ABB RobotStudio station: material handling 06 03 2024 guna basith_1.rsstn

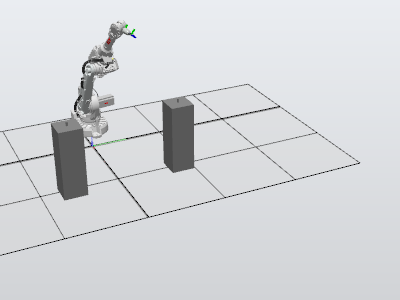
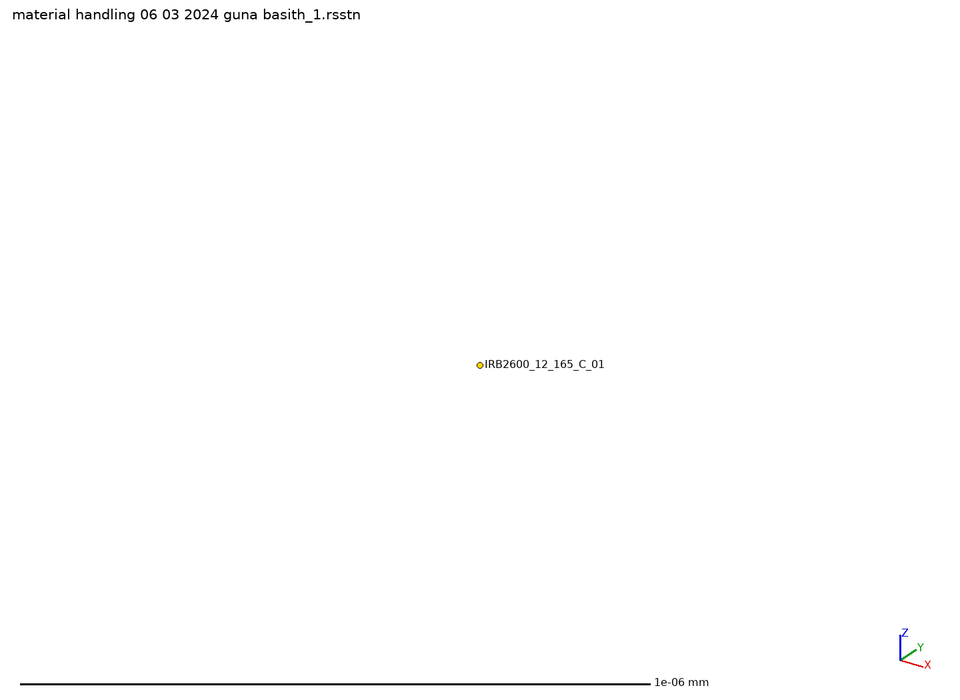
[picture v1: parts stored in the station drawn from their meshes, with robot base, taught points and paths (robot models come from the ABB library and are not in the file)]
Station Station (saved by RobotStudio 23.4.10609.1)
Controller Controller16, task T_ROB1: task frame (RAPID world) sits at (0, 0, 245) mm in the station
Controller Controller16
  mechanical unit ROB_1: IRB2600_12_165_C_01, 6 joints, base frame (0, 0, 0) mm
Layout (positions relative to the parent item):
  - Concrete [part, from Dispencing\Concrete.rslib]
  - IRB2600_12_165_C_01 [mechanism, from %ABB.RobotStudio.Models.IRB2600%\IRB2600_12_165_C_01.rslib] at (0, 0, 245) mm; joint values [0.1438, 0.4918, -1.2873, 3.4677, -1.1118, 3.9518] (rad or m)
  - SmartComponent_3 [smart component] at (1018.61, 172.16, 1931.71) mm, rotated rx 108.49 ry 28.78 rz 124.78 deg
      signals: DI attach
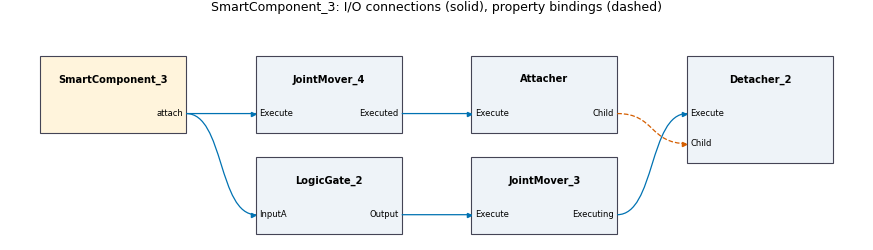
      connections:
        SmartComponent_3.attach -> JointMover_4.Execute
        JointMover_4.Executed -> Attacher.Execute
        SmartComponent_3.attach -> LogicGate_2.InputA
        LogicGate_2.Output -> JointMover_3.Execute
        JointMover_3.Executing -> Detacher_2.Execute
        Attacher.Child => Detacher_2.Child
    - Smart_Gripper_Servo_Fingers [mechanism, from %ABB.RobotStudio.Models.SmartGripper%\ABB_Smart_Gripper_Servo_Fingers.rslib] at (0, 0, 0) mm; joint values [0.023] (rad or m)
    - JointMover_3 [smart component, from Components\JointMover.rslib]
        properties: Mechanism=Smart_Gripper_Servo_Fingers; Relative=false; Duration=0; J1=0.024
    - JointMover_4 [smart component, from Components\JointMover.rslib]
        properties: Mechanism=Smart_Gripper_Servo_Fingers; Relative=false; Duration=0; J1=0.023
    - Detacher_2 [smart component, from Components\Detacher.rslib]
        properties: Child=(none); KeepPosition=true
    - Attacher [smart component, from Components\Attacher.rslib]
        properties: Parent=Smart_Gripper_Servo_Fingers; Flange=0; Child=(none); Mount=false; Offset=[0 0 0]; Orientation=[0 0 0]
    - LogicGate_2 [smart component, from Components\LogicGate.rslib]
        properties: Operator=NOT; Delay=0
  - table1 [part] at (870, 684.21, 0) mm, size 300 x 300 x 900 mm
  - table2 [part] at (914.65, -761.84, 0) mm, size 300 x 300 x 900 mm
  - object [part] at (1020, 834.21, 900) mm, size 24 x 23.9 x 50 mm
  - object2 [part] at (1064.65, -611.84, 900) mm, size 24 x 23.9 x 50 mm
Attachment: SmartComponent_3 is attached to IRB2600_12_165_C_01 / Link6
Targets, tools, work objects and paths stored in the station, written as RAPID:
! task T_ROB1
MODULE CalibData
  PERS tooldata Servo:=[TRUE,[[0,0,114.2],[1,0,0,0]],[0.215,[8.7,12.3,49.2],[1,0,0,0],0.00021,0.00024,0.00009]];
ENDMODULE

